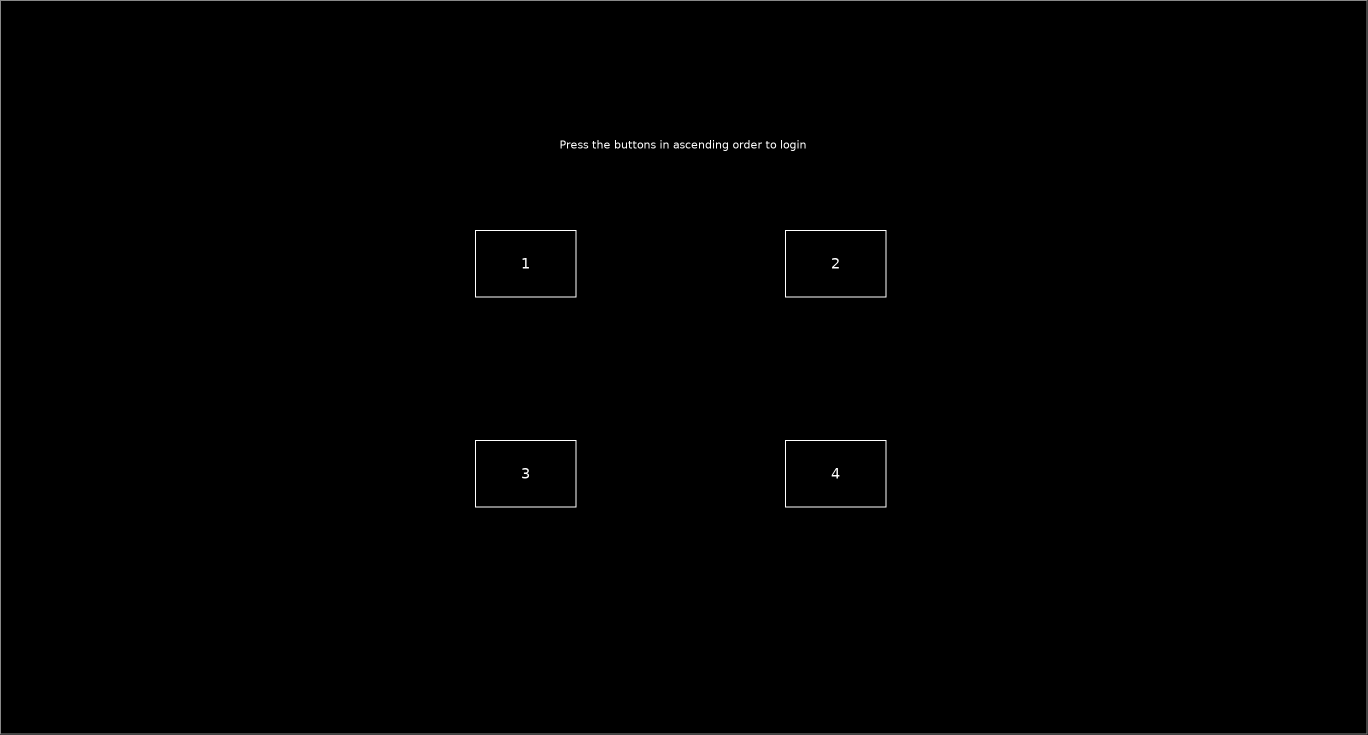
VISUALIZATION VISU_MTCSBlankScreen  // 1368x735
    Rectangle (0,-35 1366x768)
        OnMouseClick: execute { GLOBAL.gui.blankScreen.do_anywhere := TRUE; }
    Rectangle (475,230 101x67), "1", invisible if: GLOBAL.gui.blankScreen.totallyBlank
        OnMouseClick: execute { GLOBAL.gui.blankScreen.do_1 := TRUE; }
    Rectangle (785,230 101x67), "2", invisible if: GLOBAL.gui.blankScreen.totallyBlank
        OnMouseClick: execute { GLOBAL.gui.blankScreen.do_2 := TRUE; }
    Rectangle (475,440 101x67), "3", invisible if: GLOBAL.gui.blankScreen.totallyBlank
        OnMouseClick: execute { GLOBAL.gui.blankScreen.do_3 := TRUE; }
    Rectangle (785,440 101x67), "4", invisible if: GLOBAL.gui.blankScreen.totallyBlank, input disabled if: GLOBAL.gui.blankScreen.deactivate_4
        OnMouseClick: change screen: VISU_MAIN
    Label (405,130 556x30), "Press the buttons in ascending order to login", invisible if: GLOBAL.gui.blankScreen.totallyBlank
END_VISUALIZATION

(* stored: Version 1.1.0.1, ProductVersion 3.1.4018.5
   Visu VISU_MTCSBlankScreen: Id {c7cd01d6-32a1-44d4-97b5-5f6d32cbe937} *)
